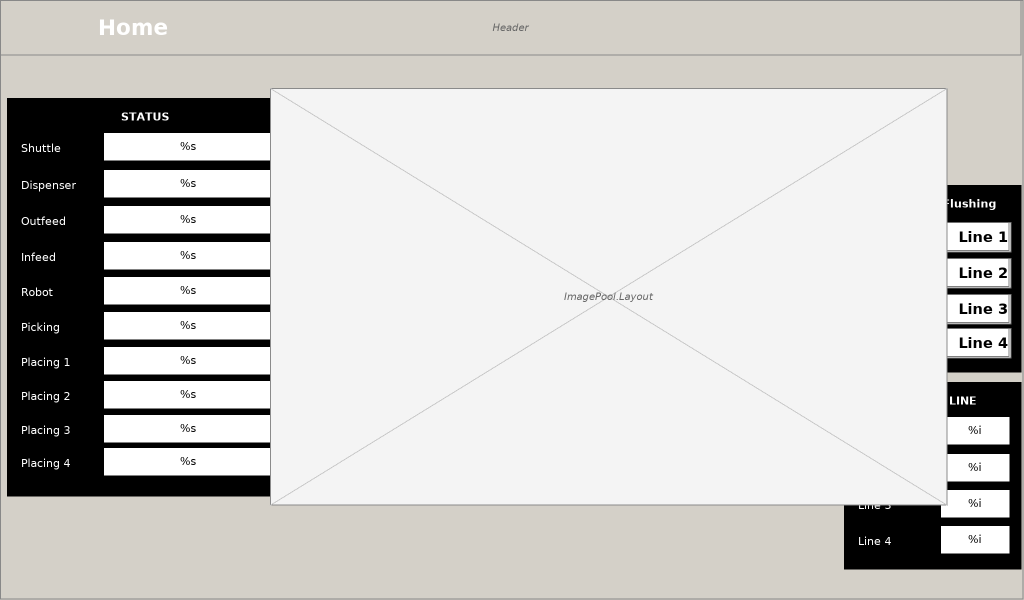
VISUALIZATION Home  // 1024x600
    RoundedRectangle (917,185 104x187)
    Frame (0,0 1021x55)
        shows Header()
    Label (95,15 214x25), "Home"
    RoundedRectangle (844,382 177x187)
    Label (869,381 125x40), "COUNTER LINE"
    Label (855,415 78x35), "Line 1"
    RoundedRectangle (940,416 70x29), "%i", text variable: HMI_GVL.arCountReal[1], input disabled if: Data_GVL.stStateMachineRobot.Running
        OnMouseClick: write the text variable via Default
    Label (855,452 78x35), "Line 2"
    RoundedRectangle (940,453 70x29), "%i", text variable: HMI_GVL.arCountReal[2], input disabled if: Data_GVL.stStateMachineRobot.Running
        OnMouseClick: write the text variable via Default
    Label (855,488 78x35), "Line 3"
    RoundedRectangle (940,489 70x29), "%i", text variable: HMI_GVL.arCountReal[3], input disabled if: Data_GVL.stStateMachineRobot.Running
        OnMouseClick: write the text variable via Default
    Label (855,524 78x35), "Line 4"
    RoundedRectangle (940,525 70x29), "%i", text variable: HMI_GVL.arCountReal[4], input disabled if: Data_GVL.stStateMachineRobot.Running
        OnMouseClick: write the text variable via Default
    Group (7,97 279x399)
        RoundedRectangle (0,1 279x398)
        Label (25,0 227x40), "STATUS"
        Label (11,34 78x35), "Shuttle"
        RoundedRectangle (96,35 170x29), "%s", text variable: InputOutput_GVL.Shuttle_stsMachine
        Label (11,71 78x35), "Dispenser"
        RoundedRectangle (96,72 170x29), "%s", text variable: InputOutput_GVL.Dispenser_stsMachine
        Label (11,107 78x35), "Outfeed"
        RoundedRectangle (96,108 170x29), "%s", text variable: InputOutput_GVL.Outfeed_stsMachine
        Label (11,143 78x35), "Infeed"
        RoundedRectangle (96,144 170x29), "%s", text variable: InputOutput_GVL.Infeed_stsMachine
        Label (11,178 78x35), "Robot"
        RoundedRectangle (96,179 170x29), "%s", text variable: Data_GVL.StateMachineRobot_stsMachine
        Label (11,213 78x35), "Picking"
        RoundedRectangle (96,214 170x29), "%s", text variable: Data_GVL.StateMachinePicking_stsMachine
        Label (11,248 78x35), "Placing 1"
        RoundedRectangle (96,249 170x29), "%s", text variable: Data_GVL.StateMachinePlacing1_stsMachine
        Label (11,282 78x35), "Placing 2"
        RoundedRectangle (96,283 170x29), "%s", text variable: Data_GVL.StateMachinePlacing2_stsMachine
        Label (11,316 78x35), "Placing 3"
        RoundedRectangle (96,317 170x29), "%s", text variable: Data_GVL.StateMachinePlacing3_stsMachine
        Label (11,349 78x35), "Placing 4"
        RoundedRectangle (96,350 170x29), "%s", text variable: Data_GVL.StateMachinePlacing4_stsMachine
    Button (930,222 81x30), "Line 1", image: VisuSymbols.Symbols.Rec
        tap HMI_GVL.Flush_Placing1
    Label (907,184 125x40), "Flushing"
    Button (930,258 81x30), "Line 2", image: VisuSymbols.Symbols.Rec
        tap HMI_GVL.Flush_Placing2
    Button (930,294 81x30), "Line 3", image: VisuSymbols.Symbols.Rec
        tap HMI_GVL.Flush_Placing3
    Button (930,328 81x30), "Line 4", image: VisuSymbols.Symbols.Rec
        tap HMI_GVL.Flush_Placing4
    Image (270,88 677x417), image: ImagePool.Layout
END_VISUALIZATION

(* stored: Version 1.1.0.1, ProductVersion 3.1.4024.12
   Visu Home: Id {e26e06b9-3998-42dc-b55e-65186601207d} *)
